(* IEC 61131-3 sources: TA/Tests/SampleBuffer, 6 files *)

(* ---- varGenerator.st ---- *)
FUNCTION_BLOCK varGenerator

IF CntGenerator = currentCntGenerator OR NOT StartGenerator THEN
    varOut_BOOL := FALSE;
    varOut_BYTE := 0;
    varOut_DATE := ANY_TO_DATE(0);
    varOut_DINT := 0;
    varOut_DWORD := 0;
    varOut_INT := 0;
    varOut_LINT := 0;
    varOut_LREAL := 0;
    varOut_LWORD := 0;
    varOut_REAL := 0;
    varOut_SINT := 0;
    varOut_STRING := ' ';
    varOut_TIME := T#0ms;
    varOut_UDINT := 0;
    varOut_UINT := 0;
    varOut_ULINT := 0;
    varOut_USINT := 0;
    varOut_WORD := 0;

    StartGenerator := FALSE;
    currentCntGenerator := 0;
    FinalGenerating := FALSE;
END_IF;

IF StartGenerator THEN
    currentTimeGenerator := currentTimeGenerator + resCycleTime;

    IF currentTimeGenerator >= PulseTimeGenerator THEN
        varOut_BOOL := NOT varOut_BOOL;
        varOut_BYTE := varOut_BYTE + 1;
        varOut_DATE := ANY_TO_DATE(1445385600 + varOut_DINT * 86400);
        varOut_DINT := varOut_DINT + 1;
        varOut_DWORD := varOut_DWORD + 1;
        varOut_INT :=varOut_INT + 1;
        varOut_LINT := varOut_LINT + 1;
        varOut_LREAL := ANY_TO_LREAL(varOut_LINT) / 100;
        varOut_LWORD := varOut_LWORD + 1;
        varOut_REAL := ANY_TO_REAL(varOut_LINT) / 10;
        varOut_SINT := varOut_SINT + 1;
        varOut_STRING := ANY_TO_STRING(varOut_DINT) + ' ' + ANY_TO_STRING(varOut_TIME);
        varOut_TIME := varOut_TIME + PulseTimeGenerator;
        varOut_UDINT := varOut_UDINT + 1;
        varOut_UINT := varOut_UINT + 1;
        varOut_ULINT := varOut_ULINT + 1;
        varOut_USINT := varOut_USINT + 1;
        varOut_WORD := varOut_WORD + 1;

        currentTimeGenerator := T#0ms;
        currentCntGenerator := currentCntGenerator + 1;

        IF CntGenerator = currentCntGenerator THEN
            FinalGenerating := TRUE;
        END_IF;
    END_IF;
END_IF;

END_FUNCTION_BLOCK

(* ---- varGenerator_CPU850.st ---- *)
FUNCTION_BLOCK varGenerator_CPU850

IF CntGenerator = currentCntGenerator OR NOT StartGenerator THEN
    varOut_BOOL := FALSE;
    varOut_BYTE := 0;
    varOut_DINT := 0;
    varOut_DWORD := 0;
    varOut_INT := 0;
    varOut_LINT := 0;
    varOut_LREAL := 0;
    varOut_LWORD := 0;
    varOut_REAL := 0;
    varOut_SINT := 0;
    varOut_TIME := T#0ms;
    varOut_UDINT := 0;
    varOut_UINT := 0;
    varOut_ULINT := 0;
    varOut_USINT := 0;
    varOut_WORD := 0;

    StartGenerator := FALSE;
    currentCntGenerator := 0;
    FinalGenerating := FALSE;
END_IF;

IF StartGenerator THEN
    currentTimeGenerator := currentTimeGenerator + resCycleTime;

    IF currentTimeGenerator >= PulseTimeGenerator THEN
        varOut_BOOL := NOT varOut_BOOL;
        varOut_LINT := varOut_LINT + 1;
        varOut_TIME := varOut_TIME + PulseTimeGenerator;

        varOut_BYTE := ANY_TO_BYTE(varOut_LINT);
        varOut_DINT := ANY_TO_DINT(varOut_LINT);
        varOut_DWORD := ANY_TO_DWORD(varOut_LINT);
        varOut_INT := ANY_TO_INT(varOut_LINT);
        varOut_LREAL := ANY_TO_LREAL(varOut_LINT) / 100;
        varOut_LWORD := ANY_TO_LWORD(varOut_LINT);
        varOut_REAL := ANY_TO_REAL(varOut_LINT) / 10;
        varOut_SINT := ANY_TO_SINT(varOut_LINT);
        varOut_UDINT := ANY_TO_UDINT(varOut_LINT);
        varOut_UINT := ANY_TO_UINT(varOut_LINT);
        varOut_ULINT := ANY_TO_ULINT(varOut_LINT);
        varOut_USINT := ANY_TO_USINT(varOut_LINT);
        varOut_WORD := ANY_TO_WORD(varOut_LINT);

        currentTimeGenerator := T#0ms;
        currentCntGenerator := currentCntGenerator + 1;

        IF CntGenerator = currentCntGenerator THEN
            FinalGenerating := TRUE;
        END_IF;
    END_IF;
END_IF;

END_FUNCTION_BLOCK

(* ---- SampleBuffer_CPU715.st ---- *)
PROGRAM SampleBuffer

CurrentCycleTime := __SYSVA_TCYCYCTIME;

testBufferGenerator.StartGenerator := StartSampleBufferTest;
testBufferGenerator.CntGenerator := CntSampleBufferTest;
testBufferGenerator.PulseTimeGenerator := PulseTimeSampleBufferTest;
testBufferGenerator.resCycleTime := __SYSVA_TCYCYCTIME;
testBufferGenerator(.StartGenerator, .CntGenerator, .PulseTimeGenerator, .resCycleTime);

SampleBuffer_BOOL := testBufferGenerator.varOut_BOOL;
SampleBuffer_BYTE := testBufferGenerator.varOut_BYTE;
SampleBuffer_DATE := testBufferGenerator.varOut_DATE;
SampleBuffer_DINT := testBufferGenerator.varOut_DINT;
SampleBuffer_DWORD := testBufferGenerator.varOut_DWORD;
SampleBuffer_INT := testBufferGenerator.varOut_INT;
SampleBuffer_LINT := testBufferGenerator.varOut_LINT;
SampleBuffer_LREAL := testBufferGenerator.varOut_LREAL;
SampleBuffer_LWORD := testBufferGenerator.varOut_LWORD;
SampleBuffer_REAL := testBufferGenerator.varOut_REAL;
SampleBuffer_SINT := testBufferGenerator.varOut_SINT;
SampleBuffer_STRING := testBufferGenerator.varOut_STRING;
SampleBuffer_TIME := testBufferGenerator.varOut_TIME;
SampleBuffer_UDINT := testBufferGenerator.varOut_UDINT;
SampleBuffer_UINT := testBufferGenerator.varOut_UINT;
SampleBuffer_ULINT := testBufferGenerator.varOut_ULINT;
SampleBuffer_USINT := testBufferGenerator.varOut_USINT;
SampleBuffer_WORD := testBufferGenerator.varOut_WORD;

IF testBufferGenerator.FinalGenerating THEN
    StartSampleBufferTest := FALSE;
    CntSampleBufferTest := 0;
    PulseTimeSampleBufferTest := T#0ms;
END_IF;

END_PROGRAM

(* ---- SampleBuffer_CPU850_RT.st ---- *)
PROGRAM SampleBuffer

CurrentCycleTime_RT := _PRESET_CYCLE_TIME;

testBufferGenerator.StartGenerator := StartSampleBufferTest_RT;
testBufferGenerator.CntGenerator := CntSampleBufferTest_RT;
testBufferGenerator.PulseTimeGenerator := PulseTimeSampleBufferTest_RT;
testBufferGenerator();

SampleBuffer_BOOL_RT := testBufferGenerator.varOut_BOOL;
SampleBuffer_BYTE_RT := testBufferGenerator.varOut_BYTE;
SampleBuffer_DINT_RT := testBufferGenerator.varOut_DINT;
SampleBuffer_DWORD_RT := testBufferGenerator.varOut_DWORD;
SampleBuffer_INT_RT := testBufferGenerator.varOut_INT;
SampleBuffer_LINT_RT := testBufferGenerator.varOut_LINT;
SampleBuffer_LREAL_RT := testBufferGenerator.varOut_LREAL;
SampleBuffer_LWORD_RT := testBufferGenerator.varOut_LWORD;
SampleBuffer_REAL_RT := testBufferGenerator.varOut_REAL;
SampleBuffer_SINT_RT := testBufferGenerator.varOut_SINT;
SampleBuffer_TIME_RT := testBufferGenerator.varOut_TIME;
SampleBuffer_UDINT_RT := testBufferGenerator.varOut_UDINT;
SampleBuffer_UINT_RT := testBufferGenerator.varOut_UINT;
SampleBuffer_ULINT_RT := testBufferGenerator.varOut_ULINT;
SampleBuffer_USINT_RT := testBufferGenerator.varOut_USINT;
SampleBuffer_WORD_RT := testBufferGenerator.varOut_WORD;

IF testBufferGenerator.FinalGenerating THEN
    StartSampleBufferTest_RT := FALSE;
    CntSampleBufferTest_RT := 0;
    PulseTimeSampleBufferTest_RT := T#0ms;
END_IF;

END_PROGRAM

(* ---- SampleBuffer_CPU850_SF.st ---- *)
PROGRAM SampleBuffer

CurrentCycleTime_SF := _PRESET_CYCLE_TIME;

testBufferGenerator.StartGenerator := StartSampleBufferTest_SF;
testBufferGenerator.CntGenerator := CntSampleBufferTest_SF;
testBufferGenerator.PulseTimeGenerator := PulseTimeSampleBufferTest_SF;
testBufferGenerator();

SampleBuffer_BOOL_SF := testBufferGenerator.varOut_BOOL;
SampleBuffer_BYTE_SF := testBufferGenerator.varOut_BYTE;
SampleBuffer_DINT_SF := testBufferGenerator.varOut_DINT;
SampleBuffer_DWORD_SF := testBufferGenerator.varOut_DWORD;
SampleBuffer_INT_SF := testBufferGenerator.varOut_INT;
SampleBuffer_LINT_SF := testBufferGenerator.varOut_LINT;
SampleBuffer_LREAL_SF := testBufferGenerator.varOut_LREAL;
SampleBuffer_LWORD_SF := testBufferGenerator.varOut_LWORD;
SampleBuffer_REAL_SF := testBufferGenerator.varOut_REAL;
SampleBuffer_SINT_SF := testBufferGenerator.varOut_SINT;
SampleBuffer_TIME_SF := testBufferGenerator.varOut_TIME;
SampleBuffer_UDINT_SF := testBufferGenerator.varOut_UDINT;
SampleBuffer_UINT_SF := testBufferGenerator.varOut_UINT;
SampleBuffer_ULINT_SF := testBufferGenerator.varOut_ULINT;
SampleBuffer_USINT_SF := testBufferGenerator.varOut_USINT;
SampleBuffer_WORD_SF := testBufferGenerator.varOut_WORD;

IF testBufferGenerator.FinalGenerating THEN
    StartSampleBufferTest_SF := FALSE;
    CntSampleBufferTest_SF := 0;
    PulseTimeSampleBufferTest_SF := T#0ms;
END_IF;

END_PROGRAM

(* ---- SampleBuffer_ICORE2.st ---- *)
PROGRAM SampleBuffer

CurrentCycleTime := _PRESET_CYCLE_TIME;

testBufferGenerator.StartGenerator := StartSampleBufferTest;
testBufferGenerator.CntGenerator := CntSampleBufferTest;
testBufferGenerator.PulseTimeGenerator := PulseTimeSampleBufferTest;
testBufferGenerator.resCycleTime := _PRESET_CYCLE_TIME;
testBufferGenerator();

SampleBuffer_BOOL := testBufferGenerator.varOut_BOOL;
SampleBuffer_BYTE := testBufferGenerator.varOut_BYTE;
SampleBuffer_DATE := testBufferGenerator.varOut_DATE;
SampleBuffer_DINT := testBufferGenerator.varOut_DINT;
SampleBuffer_DWORD := testBufferGenerator.varOut_DWORD;
SampleBuffer_INT := testBufferGenerator.varOut_INT;
SampleBuffer_LINT := testBufferGenerator.varOut_LINT;
SampleBuffer_LREAL := testBufferGenerator.varOut_LREAL;
SampleBuffer_LWORD := testBufferGenerator.varOut_LWORD;
SampleBuffer_REAL := testBufferGenerator.varOut_REAL;
SampleBuffer_SINT := testBufferGenerator.varOut_SINT;
SampleBuffer_STRING := testBufferGenerator.varOut_STRING;
SampleBuffer_TIME := testBufferGenerator.varOut_TIME;
SampleBuffer_UDINT := testBufferGenerator.varOut_UDINT;
SampleBuffer_UINT := testBufferGenerator.varOut_UINT;
SampleBuffer_ULINT := testBufferGenerator.varOut_ULINT;
SampleBuffer_USINT := testBufferGenerator.varOut_USINT;
SampleBuffer_WORD := testBufferGenerator.varOut_WORD;

IF testBufferGenerator.FinalGenerating THEN
    StartSampleBufferTest := FALSE;
    CntSampleBufferTest := 0;
    PulseTimeSampleBufferTest := T#0ms;
END_IF;

END_PROGRAM
